// TIA Portal V20 export
DATA_BLOCK "AnodePnPZ1ReelCutDataDeleteOn"   // DB134, Motion_DB
// stored: InstanceOfName TO_OutputCam, OfSystemLibElement TO_OutputCam, OfSystemLibVersion 9.0
TO_OutputCam   // technology object, version 9.0
   // // inherited from TO_Object
   // VAR
   //    CamOutput { ExternalWritable := 'False'} : Bool;
   //    Parameter { S7_SetPoint := 'True'} : TO_OutputCam_Struct_Parameter;
   //    Interface { S7_SetPoint := 'True'} : TO_OutputCam_Struct_Interface;
   //    Units { ExternalWritable := 'False'; S7_SetPoint := 'True'} : TO_OutputCam_Struct_Units;
   //    StatusWord { ExternalWritable := 'False'} : DWord;
   //    ErrorWord { ExternalWritable := 'False'} : DWord;
   //    ErrorDetail { ExternalWritable := 'False'; S7_SetPoint := 'True'} : TO_Struct_ErrorDetail;
   //    WarningWord { ExternalWritable := 'False'} : DWord;
   // END_VAR
BEGIN
END_DATA_BLOCK
